PROGRAM PnpCtrl_Arm1

VAR
	fbArmPnpCtrl_Arm1		: fbV2_ArmPnpCtrl;

	fbArmPnpCtrl_Arm1a		: fbV2_1_ArmPnpCtrl;

	Arm1Agi: fbArmSpecialFunctionStore;

	fbVertAgiMovement: fbAxisAgiMovement;

END_VAR

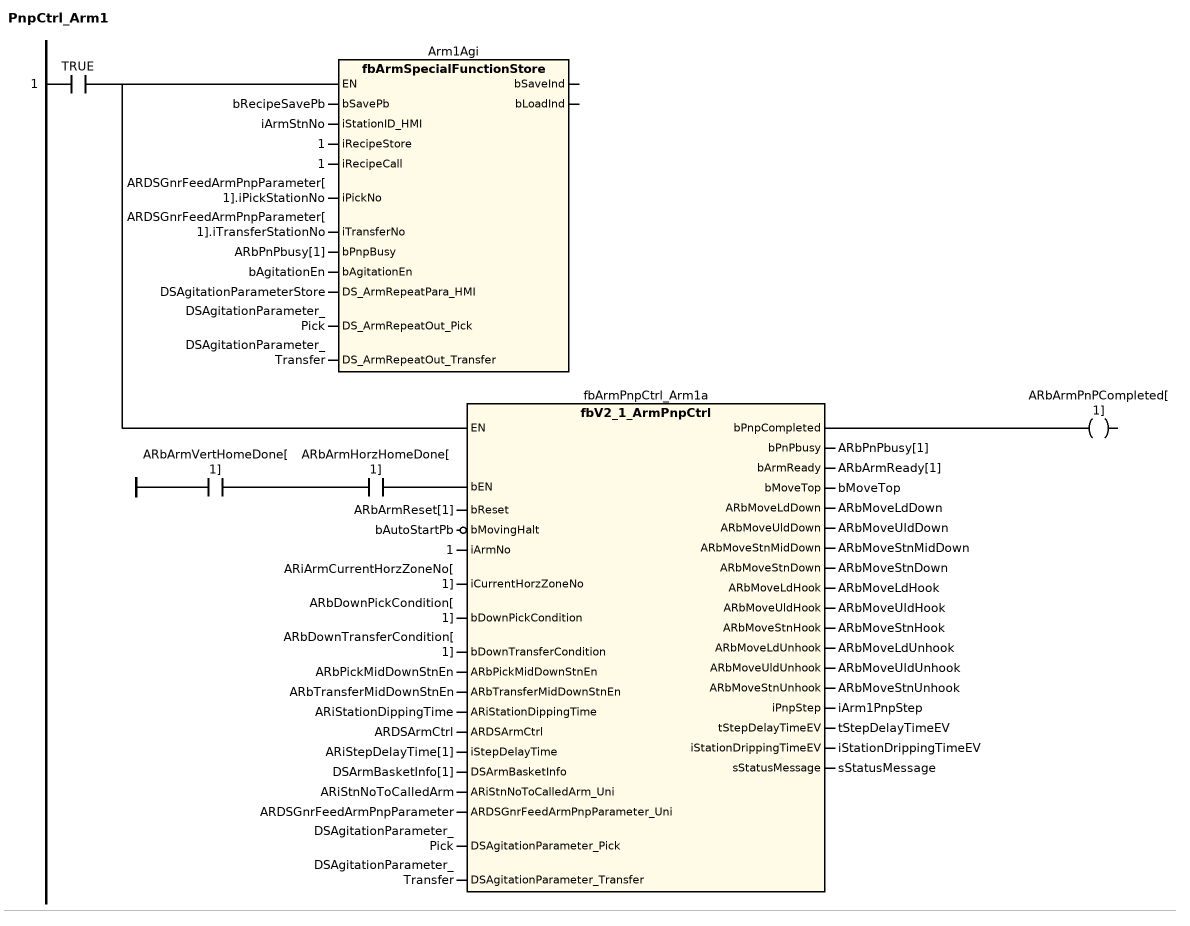
// NETWORK 1
Arm1Agi(
    bSavePb := bRecipeSavePb,
    iStationID_HMI := iArmStnNo,
    iRecipeStore := 1,
    iRecipeCall := 1,
    iPickNo := ARDSGnrFeedArmPnpParameter[1].iPickStationNo,
    iTransferNo := ARDSGnrFeedArmPnpParameter[1].iTransferStationNo,
    bPnpBusy := ARbPnPbusy[1],
    bAgitationEn := bAgitationEn,
    DS_ArmRepeatPara_HMI := DSAgitationParameterStore,
    DS_ArmRepeatOut_Pick := DSAgitationParameter_Pick,
    DS_ArmRepeatOut_Transfer := DSAgitationParameter_Transfer); // fbArmSpecialFunctionStore
fbArmPnpCtrl_Arm1a(
    bEN := ARbArmVertHomeDone[1] AND ARbArmHorzHomeDone[1],
    bReset := ARbArmReset[1],
    bMovingHalt := NOT bAutoStartPb,
    iArmNo := 1,
    iCurrentHorzZoneNo := ARiArmCurrentHorzZoneNo[1],
    bDownPickCondition := ARbDownPickCondition[1],
    bDownTransferCondition := ARbDownTransferCondition[1],
    ARbPickMidDownStnEn := ARbPickMidDownStnEn,
    ARbTransferMidDownStnEn := ARbTransferMidDownStnEn,
    ARiStationDippingTime := ARiStationDippingTime,
    ARDSArmCtrl := ARDSArmCtrl,
    iStepDelayTime := ARiStepDelayTime[1],
    DSArmBasketInfo := DSArmBasketInfo[1],
    ARiStnNoToCalledArm_Uni := ARiStnNoToCalledArm,
    ARDSGnrFeedArmPnpParameter_Uni := ARDSGnrFeedArmPnpParameter,
    DSAgitationParameter_Pick := DSAgitationParameter_Pick,
    DSAgitationParameter_Transfer := DSAgitationParameter_Transfer,
    bPnPbusy => ARbPnPbusy[1],
    bArmReady => ARbArmReady[1],
    bMoveTop => bMoveTop,
    ARbMoveLdDown => ARbMoveLdDown,
    ARbMoveUldDown => ARbMoveUldDown,
    ARbMoveStnMidDown => ARbMoveStnMidDown,
    ARbMoveStnDown => ARbMoveStnDown,
    ARbMoveLdHook => ARbMoveLdHook,
    ARbMoveUldHook => ARbMoveUldHook,
    ARbMoveStnHook => ARbMoveStnHook,
    ARbMoveLdUnhook => ARbMoveLdUnhook,
    ARbMoveUldUnhook => ARbMoveUldUnhook,
    ARbMoveStnUnhook => ARbMoveStnUnhook,
    iPnpStep => iArm1PnpStep,
    tStepDelayTimeEV => tStepDelayTimeEV,
    iStationDrippingTimeEV => iStationDrippingTimeEV,
    sStatusMessage => sStatusMessage); // fbV2_1_ArmPnpCtrl
ARbArmPnPCompleted[1] := fbArmPnpCtrl_Arm1a.bPnpCompleted;

END_PROGRAM

(* stored: Version 1.1.0.1, ProductVersion 3.1.4024.12
   POU PnpCtrl_Arm1: Id {5cb683a3-7889-4553-91f2-112a1b1ea0ca}, SpecialFunc None *)
